// TIA Portal V19 export
TYPE "C904_STU_IF_PMP_TYPIC"
   STRUCT
      CMD { ExternalAccessible := 'False'; ExternalVisible := 'False'; ExternalWritable := 'False'} : Bool;   // Aansturing pomp (TRUE = AAN / FALSE = UIT)
      CMD_RES { ExternalAccessible := 'False'; ExternalVisible := 'False'; ExternalWritable := 'False'} : Bool;   // Reset van de latched storingen
   END_STRUCT;
END_TYPE
